TYPE IoMicroEpsilonDistanceSensor :
STRUCT
	InputMicroEpsilonDistanceSensor AT %I* : REAL;	
END_STRUCT
END_TYPE

(* stored: Version 1.1.0.1, ProductVersion 3.1.4024.12
   DUT IoMicroEpsilonDistanceSensor: Id {d1183780-6ce3-4f50-900a-90a227727926} *)
